SUBAPPLICATION SubApp (* Subapplication Type *)
  (* Standard: 61499-2 *)
  (* Version 0.0, 2012-02-28, 4DIAC-IDE, 4DIAC-Consortium *)
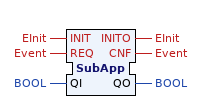
  EVENT_INPUT
    INIT : EInit; (* Initialization Request *)
    REQ; (* Normal Execution Request *)
  END_EVENT
  EVENT_OUTPUT
    INITO : EInit; (* Initialization Confirm *)
    CNF; (* Execution Confirmation *)
  END_EVENT
  VAR_INPUT
    QI : BOOL; (* Input event qualifier *)
  END_VAR
  VAR_OUTPUT
    QO : BOOL; (* Output event qualifier *)
  END_VAR
END_SUBAPPLICATION
